TYPE ST_TableNumberOut :
STRUCT
END_STRUCT
END_TYPE

(* stored: Version 1.1.0.1
   DUT ST_TableNumberOut: Id {7aab0fa3-f7d4-0c76-2b88-970dc18f8837} *)
